(* PLC project MotionTest1, Higen MCL 1 *)
(* stored: creationDateTime 2012-01-06T15:20:13, modificationDateTime 2013-03-12T12:37:18 *)

FUNCTION_BLOCK wxgetval
  VAR
    getpy : python_gear;
    latch : SR;
  END_VAR
  VAR_INPUT
    name : STRING;
  END_VAR
  VAR_OUTPUT
    val : BOOL;
  END_VAR
  VAR  (* added by the conversion: wires and edge detectors of the diagram *)
    _EQ41_ENO : BOOL;
    _EQ41_OUT : BOOL;
    _EQ3_ENO : BOOL;
    _EQ3_OUT : BOOL;
  END_VAR

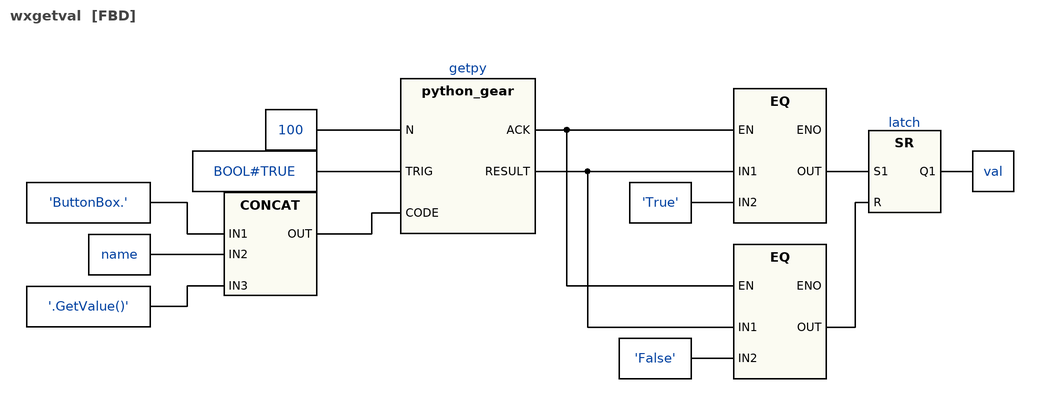
(* FBD diagram, written out as Structured Text *)
getpy(N := 100, TRIG := BOOL#TRUE, CODE := CONCAT('ButtonBox.', name, '.GetValue()'));
_EQ41_OUT := EQ(EN := getpy.ACK, IN1 := getpy.RESULT, IN2 := 'True', ENO => _EQ41_ENO);
_EQ3_OUT := EQ(EN := getpy.ACK, IN1 := getpy.RESULT, IN2 := 'False', ENO => _EQ3_ENO);
latch(S1 := _EQ41_OUT, R := _EQ3_OUT);
val := latch.Q1;
END_FUNCTION_BLOCK

PROGRAM main
  VAR
    Done : BOOL;
    Axis : AXIS_REF;
    switch : MC_Power;
    readpos : MC_ReadActualPosition;
    Pn : LREAL;
    Vn : LREAL;
    setpos : MC_SetPosition;
    readspeed : MC_ReadParameter;
    moveB : MC_Stop;
    sim : MC_Sim;
    bt1 : wxgetval;
    Block1 : wxgetval;
    Block2 : wxgetval;
    Block3 : wxgetval;
    rset : MC_Reset;
    prof : MC_PositionProfile;
    p1 : MC_WriteParameter;
    Block5 : MC_WriteParameter;
    Block6 : wxgetval;
    Block4 : wxgetval;
    Block7 : wxgetval;
    Block9 : MC_VelocityProfile;
    Block11 : MC_AccelerationProfile;
    MC_TP_REF_FROM_CSV0 : MC_TP_REF_FROM_CSV;
    MC_TV_REF_FROM_CSV0 : MC_TV_REF_FROM_CSV;
    MC_TA_REF_FROM_CSV0 : MC_TA_REF_FROM_CSV;
  END_VAR
  VAR  (* added by the conversion: wires and edge detectors of the diagram *)
    _SEL66_OUT : REAL;
    _SEL72_OUT : REAL;
    _SEL83_OUT : REAL;
  END_VAR

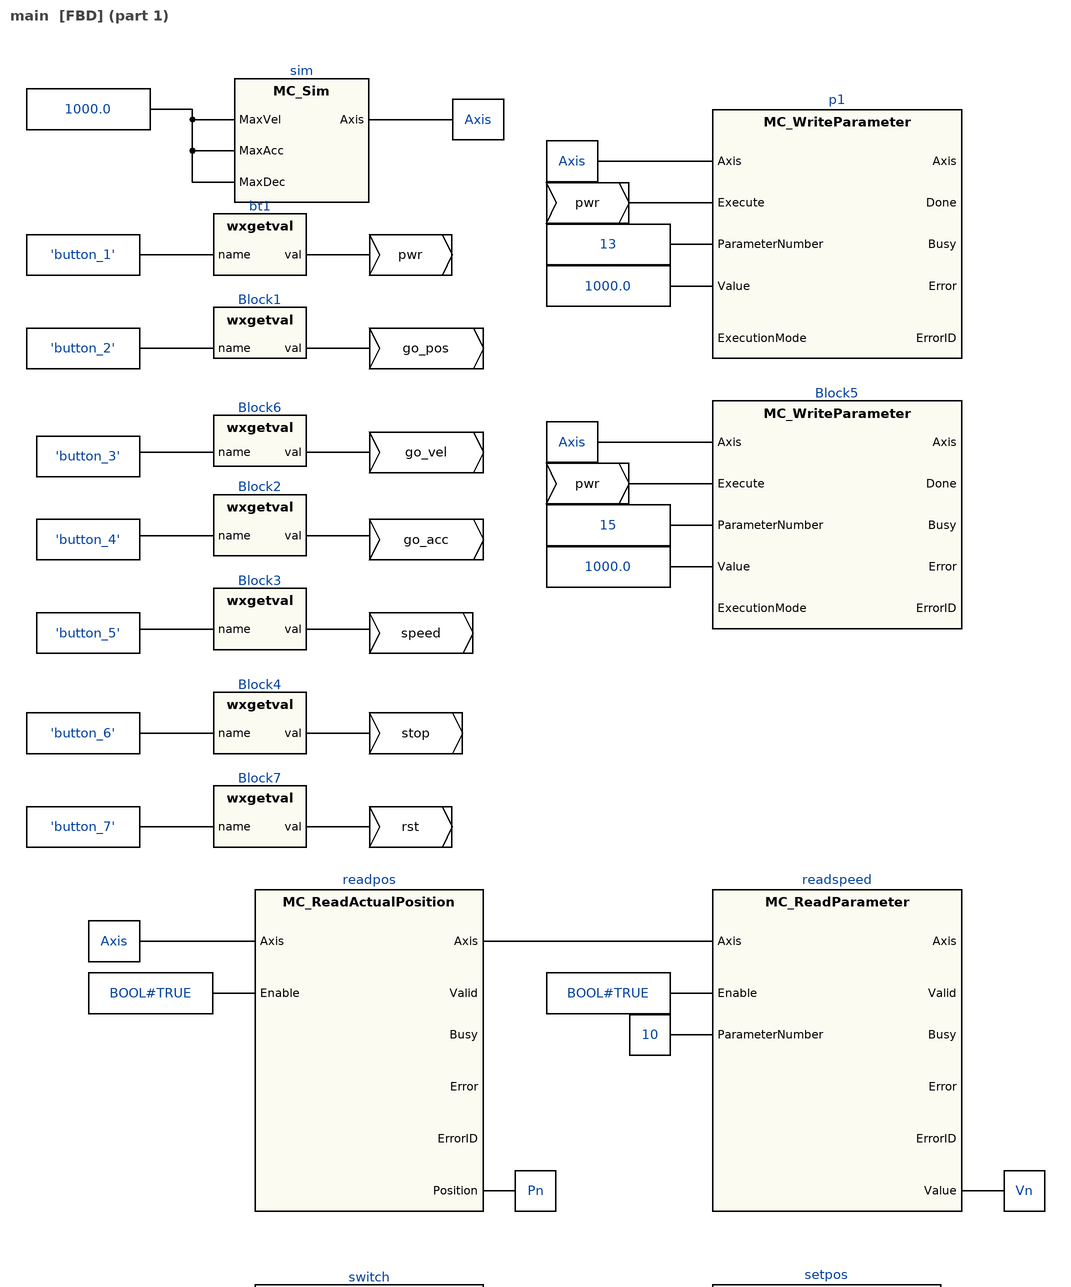
(* FBD diagram, written out as Structured Text *)
sim(MaxVel := 1000.0, MaxAcc := 1000.0, MaxDec := 1000.0);
Axis := sim.Axis;
readpos(Axis := Axis, Enable := BOOL#TRUE);
Pn := readpos.Position;
readspeed(Axis := readpos.Axis, Enable := BOOL#TRUE, ParameterNumber := 10);
Vn := readspeed.Value;
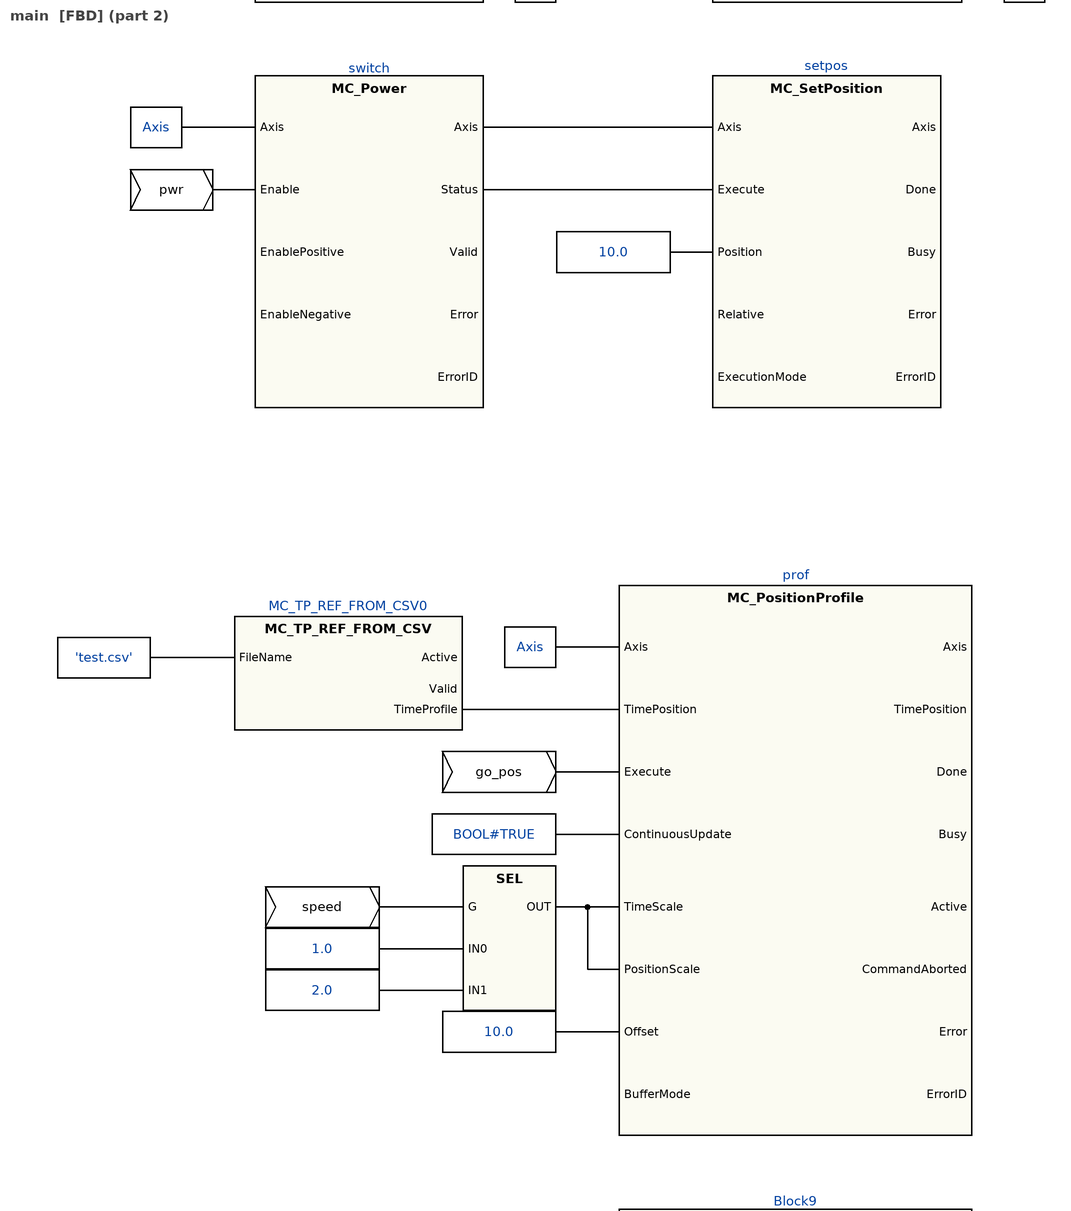
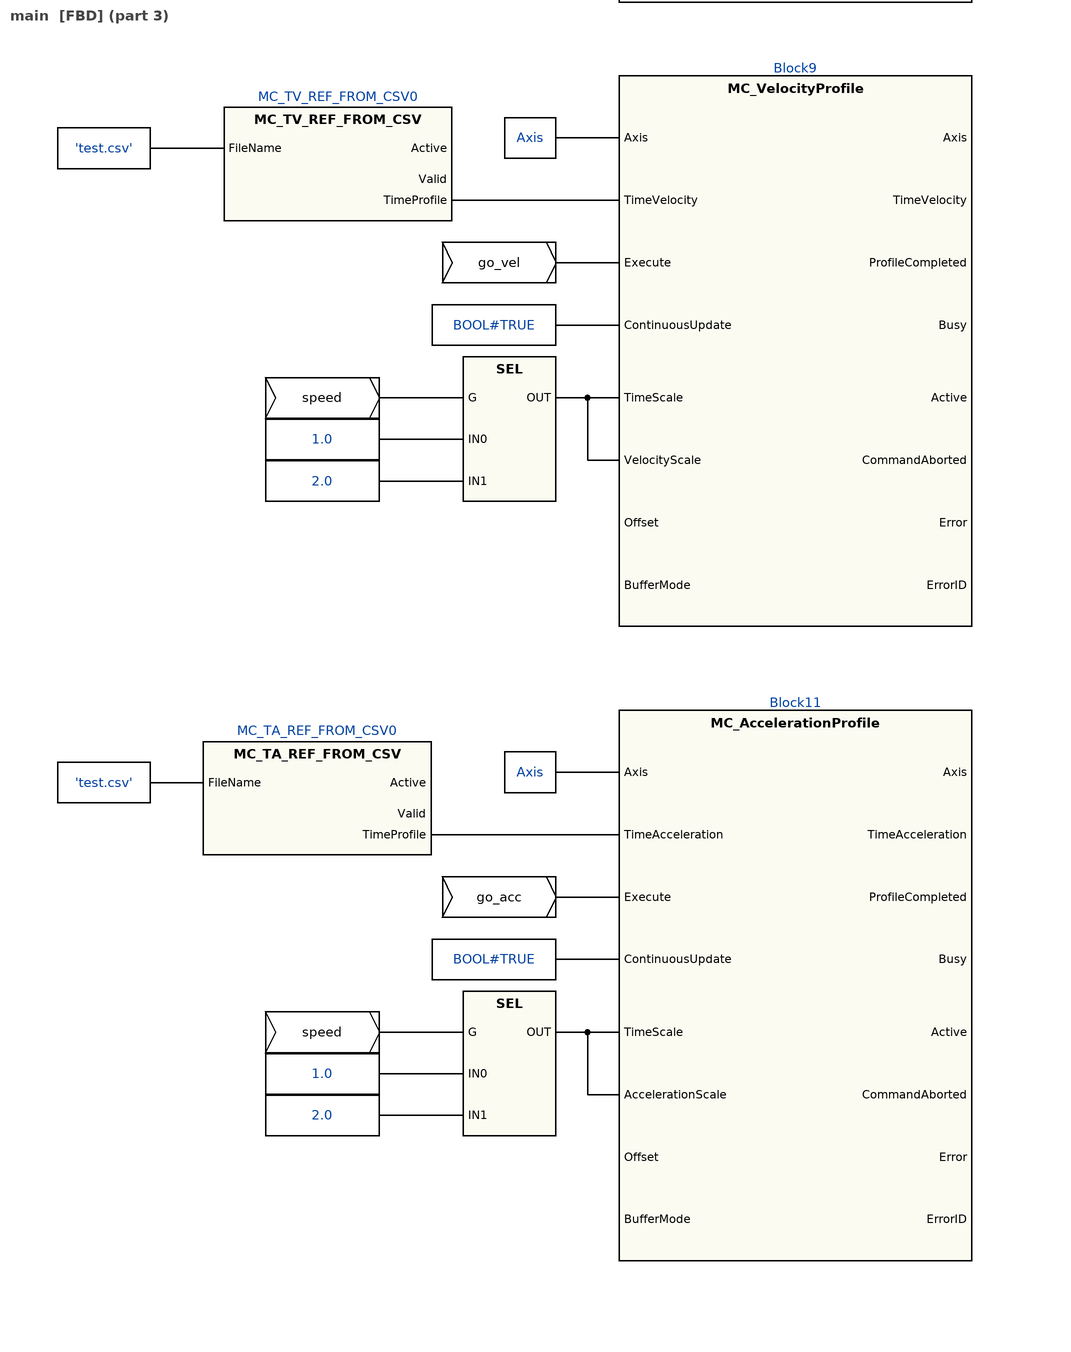
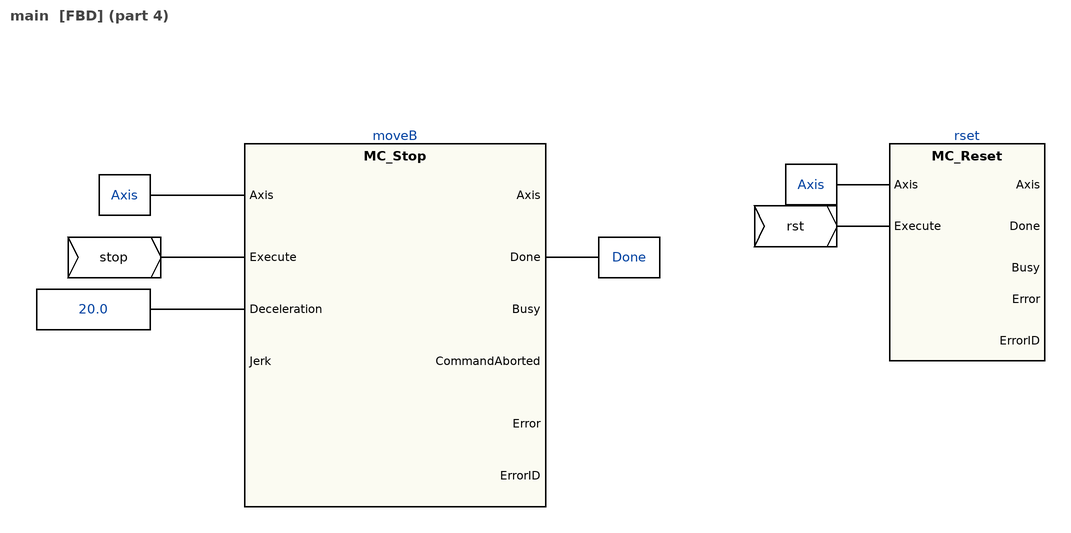
Block4(name := 'button_6');
moveB(Axis := Axis, Execute := Block4.val, Deceleration := 20.0);
Done := moveB.Done;
bt1(name := 'button_1');
p1(Axis := Axis, Execute := bt1.val, ParameterNumber := 13, Value := 1000.0);
Block1(name := 'button_2');
Block5(Axis := Axis, Execute := bt1.val, ParameterNumber := 15, Value := 1000.0);
Block6(name := 'button_3');
Block2(name := 'button_4');
Block3(name := 'button_5');
Block7(name := 'button_7');
switch(Axis := Axis, Enable := bt1.val);
setpos(Axis := switch.Axis, Execute := switch.Status, Position := 10.0);
MC_TP_REF_FROM_CSV0(FileName := 'test.csv');
_SEL66_OUT := SEL(Block3.val, 1.0, 2.0);
prof(Axis := Axis, TimePosition := MC_TP_REF_FROM_CSV0.TimeProfile, Execute := Block1.val, ContinuousUpdate := BOOL#TRUE, TimeScale := _SEL66_OUT, PositionScale := _SEL66_OUT, Offset := 10.0);
MC_TV_REF_FROM_CSV0(FileName := 'test.csv');
_SEL72_OUT := SEL(Block3.val, 1.0, 2.0);
Block9(Axis := Axis, TimeVelocity := MC_TV_REF_FROM_CSV0.TimeProfile, Execute := Block6.val, ContinuousUpdate := BOOL#TRUE, TimeScale := _SEL72_OUT, VelocityScale := _SEL72_OUT);
MC_TA_REF_FROM_CSV0(FileName := 'test.csv');
_SEL83_OUT := SEL(Block3.val, 1.0, 2.0);
Block11(Axis := Axis, TimeAcceleration := MC_TA_REF_FROM_CSV0.TimeProfile, Execute := Block2.val, ContinuousUpdate := BOOL#TRUE, TimeScale := _SEL83_OUT, AccelerationScale := _SEL83_OUT);
rset(Axis := Axis, Execute := Block7.val);
END_PROGRAM

CONFIGURATION conf
  RESOURCE res ON PLC
    TASK milisecond(INTERVAL := T#10ms, PRIORITY := 0);
    PROGRAM maininstance WITH milisecond : main;
  END_RESOURCE
END_CONFIGURATION
